// TIA Portal V17 program export: 1 tag tables, 2 data types, 1 data blocks, 2 code blocks (in call order from the OBs), 1 instance data blocks

VAR_GLOBAL   // PLC tag table "Default tag table"
END_VAR

TYPE "udtOtherPressure"
// stored: IsFailsafeCompliant false
   STRUCT
      avaragePressure : Int;
      tripleValidationActive : Int;
      dualValidationActive : Int;
      pressure1failed : Bool;
      pressure2failed : Bool;
      pressure3failed : Bool;
      moreThen1pressureFailed : Bool;
   END_STRUCT;
END_TYPE

TYPE "udtSolenoidValve"
// stored: IsFailsafeCompliant false
   STRUCT
      scaledValeu : Int := 1;
      rawValue : Int := 2;
      rawMinimum : Int := 3;
      rawMaximum : Int := 4;
      scalledMinimum : Int := 5;
      scalledMaximium : Int := 6;
   END_STRUCT;
END_TYPE

DATA_BLOCK "dbData"   // DB2
{ S7_Optimized_Access := 'TRUE' }
VERSION : 0.1
// stored: AutoNumber true, DBAccessibleFromOPCUA true, DBAccessibleFromWebserver true, IsOnlyStoredInLoadMemory false, IsRetainMemResEnabled false, IsWriteProtectedInAS false, MemoryReserve 100
   VAR
      solenoidValve1 : "udtSolenoidValve";
      solenoidValve2 { S7_SetPoint := 'True'} : "udtSolenoidValve";
      solenoidValve3 { S7_SetPoint := 'True'} : "udtSolenoidValve";
      otherPressure { S7_SetPoint := 'True'} : "udtOtherPressure";
      value : Struct
         airInletValue : Struct
            solenoidValveOpen : Bool;
         END_STRUCT;
         drainValue : Struct
            solenoidValveOpen : Bool;
         END_STRUCT;
         bledValve : Struct
            solenoidValveOpen : Bool;
         END_STRUCT;
      END_STRUCT;
      postTestResult : Struct
         preTestCheckSequence : Struct
            pressures : Struct
               validation : Struct
                  pressure1 : Int;
                  pressure2 : Int;
                  pressure3 : Int;
                  dualValidationMode : Bool;
               END_STRUCT;
               airHoldTest : Struct
                  preDwellPeriod : Bool;
                  postDwellPeriod : Bool;
               END_STRUCT;
               drainTest : Struct
                  "0.5sPostDrainValve" : Bool;
               END_STRUCT;
            END_STRUCT;
         END_STRUCT;
         mainSequence : Struct
            pressure : Struct
               postPressurizationPeriod : Bool;
               postDwellPeriod : Bool;
               bleedInterval1 : Bool;
               bleedInterval2 : Bool := false;
               bleedInterval3 : Bool := false;
               bleedInterval4 : Bool := false;
               bleedInterval5 : Bool := false;
               bleedInterval6 : Bool := false;
               bleedInterval7 : Bool := false;
               bleedInterval8 : Bool := false;
               bleedInterval9 : Bool := false;
               bleedInterval10 : Bool := false;
               bleedInterval11 : Bool := false;
               bleedInterval12 : Bool := false;
               mechanicalFailsavePressure : Bool;
            END_STRUCT;
         END_STRUCT;
      END_STRUCT;
      sequenceControl : Struct
         "startPre-TestSequecne" : Bool;
         startMainSequence : Bool;
         startSensorValidation : Bool;
         endSensorValidation : Bool;
         ActiveSequenceComplete : Bool;
         activeSequenceFailed : Bool;
         preTestSequenceActive : Bool;
         mainSequenceActive : Bool;
      END_STRUCT;
   END_VAR
BEGIN
END_DATA_BLOCK

ORGANIZATION_BLOCK "Main"   // OB1, LAD, ProgramCycle
TITLE = "Main Program Sweep (Cycle)"
{ S7_Optimized_Access := 'TRUE' }
VERSION : 0.1
// stored: AutoNumber true, IsIECCheckEnabled false, SetENOAutomatically false
   VAR_INPUT
      Initial_Call : Bool;   // Initial call of this OB
      Remanence : Bool;   // =True, if remanent data are available
   END_VAR
BEGIN
END_ORGANIZATION_BLOCK

FUNCTION_BLOCK "Main_Safety_RTG1"   // FB1, F_FBD
{ S7_Optimized_Access := 'TRUE' }
VERSION : 0.1
// stored: AutoNumber false, IsIECCheckEnabled false, UDAEnableTagReadback false
BEGIN
END_FUNCTION_BLOCK

DATA_BLOCK "Main_Safety_RTG1_DB"   // DB1, F_DB
NAME : FUSI
VERSION : 0.1
// stored: AutoNumber true, DBAccessibleFromOPCUA true, DBAccessibleFromWebserver true, InstanceOfName Main_Safety_RTG1, InstanceOfType FB
"Main_Safety_RTG1"
BEGIN
END_DATA_BLOCK
